TYPE "BTrk_item"
VERSION : 0.1
// Block: BTrk_item
   STRUCT
      B_ID : DInt;
      O_ID : DInt;
      Quality : Int;
      BLen_Meas : Real;
      W_A : Real;
      H_B : Real;
      P_L : Struct
         P_ID : DInt;
         C_ID : DInt;
         Quality : Int;
         PLen_Meas : Real;
      END_STRUCT;
      P_U : Struct
         P_ID : DInt;
         C_ID : DInt;
         Quality : Int;
         PLen_Meas : Real;
      END_STRUCT;
   END_STRUCT;

END_TYPE
